(* Visualisation VIS_CHONOEDITOR
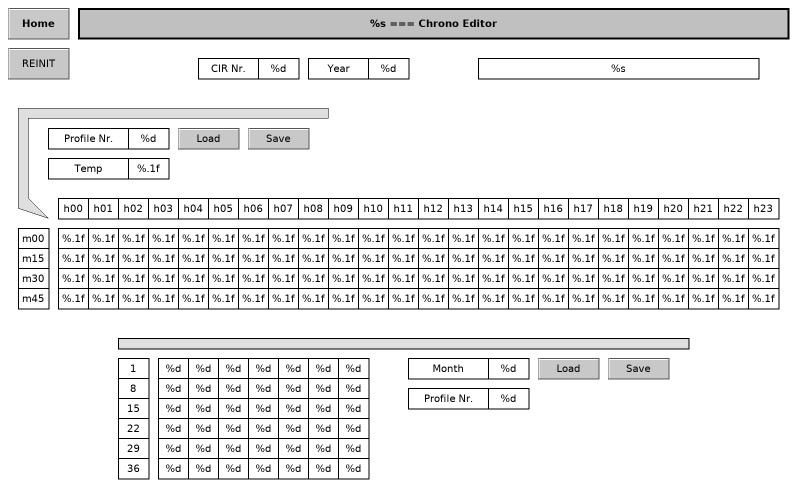
rectangle at (200,60)-(261,81): text "CIR Nr."
rectangle at (260,60)-(301,81): text "%d"; shows CronEd.CN_Sel; alarm colour if CronEd.CN_Sel<>CronEd.CN_Act; editable 1..6
rectangle at (50,130)-(131,151): text "Profile Nr."
rectangle at (130,130)-(171,151): text "%d"; shows CronEd.PR_Sel; alarm colour if CronEd.PR_Sel<>CronEd.PR_Act; editable 1..10
rectangle at (50,160)-(131,181): text "Temp"
rectangle at (130,160)-(171,181): text "%.1f"; shows CronEd.PR_TT; editable
button at (180,130)-(241,151): text "Load"; toggles CronEd.PR_Load
button at (250,130)-(311,151): text "Save"; toggles CronEd.PR_Save
rectangle at (20,230)-(51,251): text "m00"
rectangle at (20,250)-(51,271): text "m15"
rectangle at (20,270)-(51,291): text "m30"
rectangle at (20,290)-(51,311): text "m45"
rectangle at (80,10)-(791,41): text "%s === Chrono Editor"; shows .Plant_NAME
button at (10,10)-(71,41): text "Home"; opens PLC_VISU
rounded rectangle at (60,230)-(91,251): text "%.1f"; shows WORD_TO_REAL(CronEd.PR.Setpoint[0])/10; runs INTERN ASSIGN CronEd.PR.Setpoint[0]:=(REAL_TO_WORD(CronEd.PR_TT*10))
rounded rectangle at (60,250)-(91,271): text "%.1f"; shows WORD_TO_REAL(CronEd.PR.Setpoint[1])/10; runs INTERN ASSIGN CronEd.PR.Setpoint[1]:=(REAL_TO_WORD(CronEd.PR_TT*10))
rounded rectangle at (60,270)-(91,291): text "%.1f"; shows WORD_TO_REAL(CronEd.PR.Setpoint[2])/10; runs INTERN ASSIGN CronEd.PR.Setpoint[2]:=(REAL_TO_WORD(CronEd.PR_TT*10))
rounded rectangle at (60,290)-(91,311): text "%.1f"; shows WORD_TO_REAL(CronEd.PR.Setpoint[3])/10; runs INTERN ASSIGN CronEd.PR.Setpoint[3]:=(REAL_TO_WORD(CronEd.PR_TT*10))
rectangle at (60,200)-(91,221): text "h00"; runs INTERN ASSIGN CronEd.PR.Setpoint[0]:=(REAL_TO_WORD(CronEd.PR_TT*10));INTERN ASSIGN CronEd.PR.Setpoint[1]:=(REAL_TO_WORD(CronEd.PR_TT*10));INTERN ASSIGN CronEd.PR.Setpoint[2]:=(REAL_TO_WORD(CronEd.PR_TT*10));INTERN ASSIGN CronEd.PR.Setpoint[3]:=(REAL_TO_WORD(CronEd.PR_TT*10))
rounded rectangle at (90,230)-(121,251): text "%.1f"; shows WORD_TO_REAL(CronEd.PR.Setpoint[4])/10; runs INTERN ASSIGN CronEd.PR.Setpoint[4]:=(REAL_TO_WORD(CronEd.PR_TT*10))
rounded rectangle at (90,250)-(121,271): text "%.1f"; shows WORD_TO_REAL(CronEd.PR.Setpoint[5])/10; runs INTERN ASSIGN CronEd.PR.Setpoint[5]:=(REAL_TO_WORD(CronEd.PR_TT*10))
rounded rectangle at (90,270)-(121,291): text "%.1f"; shows WORD_TO_REAL(CronEd.PR.Setpoint[6])/10; runs INTERN ASSIGN CronEd.PR.Setpoint[6]:=(REAL_TO_WORD(CronEd.PR_TT*10))
rounded rectangle at (90,290)-(121,311): text "%.1f"; shows WORD_TO_REAL(CronEd.PR.Setpoint[7])/10; runs INTERN ASSIGN CronEd.PR.Setpoint[7]:=(REAL_TO_WORD(CronEd.PR_TT*10))
rectangle at (90,200)-(121,221): text "h01"; runs INTERN ASSIGN CronEd.PR.Setpoint[4]:=(REAL_TO_WORD(CronEd.PR_TT*10));INTERN ASSIGN CronEd.PR.Setpoint[5]:=(REAL_TO_WORD(CronEd.PR_TT*10));INTERN ASSIGN CronEd.PR.Setpoint[6]:=(REAL_TO_WORD(CronEd.PR_TT*10));INTERN ASSIGN CronEd.PR.Setpoint[7]:=(REAL_TO_WORD(CronEd.PR_TT*10))
rounded rectangle at (120,230)-(151,251): text "%.1f"; shows WORD_TO_REAL(CronEd.PR.Setpoint[8])/10; runs INTERN ASSIGN CronEd.PR.Setpoint[8]:=(REAL_TO_WORD(CronEd.PR_TT*10))
rounded rectangle at (120,250)-(151,271): text "%.1f"; shows WORD_TO_REAL(CronEd.PR.Setpoint[9])/10; runs INTERN ASSIGN CronEd.PR.Setpoint[9]:=(REAL_TO_WORD(CronEd.PR_TT*10))
rounded rectangle at (120,270)-(151,291): text "%.1f"; shows WORD_TO_REAL(CronEd.PR.Setpoint[10])/10; runs INTERN ASSIGN CronEd.PR.Setpoint[10]:=(REAL_TO_WORD(CronEd.PR_TT*10))
rounded rectangle at (120,290)-(151,311): text "%.1f"; shows WORD_TO_REAL(CronEd.PR.Setpoint[11])/10; runs INTERN ASSIGN CronEd.PR.Setpoint[11]:=(REAL_TO_WORD(CronEd.PR_TT*10))
rectangle at (120,200)-(151,221): text "h02"; runs INTERN ASSIGN CronEd.PR.Setpoint[8]:=(REAL_TO_WORD(CronEd.PR_TT*10));INTERN ASSIGN CronEd.PR.Setpoint[9]:=(REAL_TO_WORD(CronEd.PR_TT*10));INTERN ASSIGN CronEd.PR.Setpoint[10]:=(REAL_TO_WORD(CronEd.PR_TT*10));INTERN ASSIGN CronEd.PR.Setpoint[11]:=(REAL_TO_WORD(CronEd.PR_TT*10))
rounded rectangle at (150,230)-(181,251): text "%.1f"; shows WORD_TO_REAL(CronEd.PR.Setpoint[12])/10; runs INTERN ASSIGN CronEd.PR.Setpoint[12]:=(REAL_TO_WORD(CronEd.PR_TT*10))
rounded rectangle at (150,250)-(181,271): text "%.1f"; shows WORD_TO_REAL(CronEd.PR.Setpoint[13])/10; runs INTERN ASSIGN CronEd.PR.Setpoint[13]:=(REAL_TO_WORD(CronEd.PR_TT*10))
rounded rectangle at (150,270)-(181,291): text "%.1f"; shows WORD_TO_REAL(CronEd.PR.Setpoint[14])/10; runs INTERN ASSIGN CronEd.PR.Setpoint[14]:=(REAL_TO_WORD(CronEd.PR_TT*10))
rounded rectangle at (150,290)-(181,311): text "%.1f"; shows WORD_TO_REAL(CronEd.PR.Setpoint[15])/10; runs INTERN ASSIGN CronEd.PR.Setpoint[15]:=(REAL_TO_WORD(CronEd.PR_TT*10))
rectangle at (150,200)-(181,221): text "h03"; runs INTERN ASSIGN CronEd.PR.Setpoint[15]:=(REAL_TO_WORD(CronEd.PR_TT*10));INTERN ASSIGN CronEd.PR.Setpoint[14]:=(REAL_TO_WORD(CronEd.PR_TT*10));INTERN ASSIGN CronEd.PR.Setpoint[13]:=(REAL_TO_WORD(CronEd.PR_TT*10));INTERN ASSIGN CronEd.PR.Setpoint[12]:=(REAL_TO_WORD(CronEd.PR_TT*10))
rounded rectangle at (180,230)-(211,251): text "%.1f"; shows WORD_TO_REAL(CronEd.PR.Setpoint[16])/10; runs INTERN ASSIGN CronEd.PR.Setpoint[16]:=(REAL_TO_WORD(CronEd.PR_TT*10))
rounded rectangle at (180,250)-(211,271): text "%.1f"; shows WORD_TO_REAL(CronEd.PR.Setpoint[17])/10; runs INTERN ASSIGN CronEd.PR.Setpoint[17]:=(REAL_TO_WORD(CronEd.PR_TT*10))
rounded rectangle at (180,270)-(211,291): text "%.1f"; shows WORD_TO_REAL(CronEd.PR.Setpoint[18])/10; runs INTERN ASSIGN CronEd.PR.Setpoint[18]:=(REAL_TO_WORD(CronEd.PR_TT*10))
rounded rectangle at (180,290)-(211,311): text "%.1f"; shows WORD_TO_REAL(CronEd.PR.Setpoint[19])/10; runs INTERN ASSIGN CronEd.PR.Setpoint[19]:=(REAL_TO_WORD(CronEd.PR_TT*10))
rectangle at (180,200)-(211,221): text "h04"; runs INTERN ASSIGN CronEd.PR.Setpoint[19]:=(REAL_TO_WORD(CronEd.PR_TT*10));INTERN ASSIGN CronEd.PR.Setpoint[18]:=(REAL_TO_WORD(CronEd.PR_TT*10));INTERN ASSIGN CronEd.PR.Setpoint[17]:=(REAL_TO_WORD(CronEd.PR_TT*10));INTERN ASSIGN CronEd.PR.Setpoint[16]:=(REAL_TO_WORD(CronEd.PR_TT*10))
rounded rectangle at (210,230)-(241,251): text "%.1f"; shows WORD_TO_REAL(CronEd.PR.Setpoint[20])/10; runs INTERN ASSIGN CronEd.PR.Setpoint[20]:=(REAL_TO_WORD(CronEd.PR_TT*10))
rounded rectangle at (210,250)-(241,271): text "%.1f"; shows WORD_TO_REAL(CronEd.PR.Setpoint[21])/10; runs INTERN ASSIGN CronEd.PR.Setpoint[21]:=(REAL_TO_WORD(CronEd.PR_TT*10))
rounded rectangle at (210,270)-(241,291): text "%.1f"; shows WORD_TO_REAL(CronEd.PR.Setpoint[22])/10; runs INTERN ASSIGN CronEd.PR.Setpoint[22]:=(REAL_TO_WORD(CronEd.PR_TT*10))
rounded rectangle at (210,290)-(241,311): text "%.1f"; shows WORD_TO_REAL(CronEd.PR.Setpoint[23])/10; runs INTERN ASSIGN CronEd.PR.Setpoint[23]:=(REAL_TO_WORD(CronEd.PR_TT*10))
rectangle at (210,200)-(241,221): text "h05"; runs INTERN ASSIGN CronEd.PR.Setpoint[23]:=(REAL_TO_WORD(CronEd.PR_TT*10));INTERN ASSIGN CronEd.PR.Setpoint[22]:=(REAL_TO_WORD(CronEd.PR_TT*10));INTERN ASSIGN CronEd.PR.Setpoint[21]:=(REAL_TO_WORD(CronEd.PR_TT*10));INTERN ASSIGN CronEd.PR.Setpoint[20]:=(REAL_TO_WORD(CronEd.PR_TT*10))
rounded rectangle at (240,230)-(271,251): text "%.1f"; shows WORD_TO_REAL(CronEd.PR.Setpoint[24])/10; runs INTERN ASSIGN CronEd.PR.Setpoint[24]:=(REAL_TO_WORD(CronEd.PR_TT*10))
rounded rectangle at (240,250)-(271,271): text "%.1f"; shows WORD_TO_REAL(CronEd.PR.Setpoint[25])/10; runs INTERN ASSIGN CronEd.PR.Setpoint[25]:=(REAL_TO_WORD(CronEd.PR_TT*10))
rounded rectangle at (240,270)-(271,291): text "%.1f"; shows WORD_TO_REAL(CronEd.PR.Setpoint[26])/10; runs INTERN ASSIGN CronEd.PR.Setpoint[26]:=(REAL_TO_WORD(CronEd.PR_TT*10))
rounded rectangle at (240,290)-(271,311): text "%.1f"; shows WORD_TO_REAL(CronEd.PR.Setpoint[27])/10; runs INTERN ASSIGN CronEd.PR.Setpoint[27]:=(REAL_TO_WORD(CronEd.PR_TT*10))
rectangle at (240,200)-(271,221): text "h06"; runs INTERN ASSIGN CronEd.PR.Setpoint[27]:=(REAL_TO_WORD(CronEd.PR_TT*10));INTERN ASSIGN CronEd.PR.Setpoint[26]:=(REAL_TO_WORD(CronEd.PR_TT*10));INTERN ASSIGN CronEd.PR.Setpoint[25]:=(REAL_TO_WORD(CronEd.PR_TT*10));INTERN ASSIGN CronEd.PR.Setpoint[24]:=(REAL_TO_WORD(CronEd.PR_TT*10))
rounded rectangle at (270,230)-(301,251): text "%.1f"; shows WORD_TO_REAL(CronEd.PR.Setpoint[28])/10; runs INTERN ASSIGN CronEd.PR.Setpoint[28]:=(REAL_TO_WORD(CronEd.PR_TT*10))
rounded rectangle at (270,250)-(301,271): text "%.1f"; shows WORD_TO_REAL(CronEd.PR.Setpoint[29])/10; runs INTERN ASSIGN CronEd.PR.Setpoint[29]:=(REAL_TO_WORD(CronEd.PR_TT*10))
rounded rectangle at (270,270)-(301,291): text "%.1f"; shows WORD_TO_REAL(CronEd.PR.Setpoint[30])/10; runs INTERN ASSIGN CronEd.PR.Setpoint[30]:=(REAL_TO_WORD(CronEd.PR_TT*10))
rounded rectangle at (270,290)-(301,311): text "%.1f"; shows WORD_TO_REAL(CronEd.PR.Setpoint[31])/10; runs INTERN ASSIGN CronEd.PR.Setpoint[31]:=(REAL_TO_WORD(CronEd.PR_TT*10))
rectangle at (270,200)-(301,221): text "h07"; runs INTERN ASSIGN CronEd.PR.Setpoint[31]:=(REAL_TO_WORD(CronEd.PR_TT*10));INTERN ASSIGN CronEd.PR.Setpoint[30]:=(REAL_TO_WORD(CronEd.PR_TT*10));INTERN ASSIGN CronEd.PR.Setpoint[29]:=(REAL_TO_WORD(CronEd.PR_TT*10));INTERN ASSIGN CronEd.PR.Setpoint[28]:=(REAL_TO_WORD(CronEd.PR_TT*10))
rounded rectangle at (300,230)-(331,251): text "%.1f"; shows WORD_TO_REAL(CronEd.PR.Setpoint[32])/10; runs INTERN ASSIGN CronEd.PR.Setpoint[32]:=(REAL_TO_WORD(CronEd.PR_TT*10))
rounded rectangle at (300,250)-(331,271): text "%.1f"; shows WORD_TO_REAL(CronEd.PR.Setpoint[33])/10; runs INTERN ASSIGN CronEd.PR.Setpoint[33]:=(REAL_TO_WORD(CronEd.PR_TT*10))
rounded rectangle at (300,270)-(331,291): text "%.1f"; shows WORD_TO_REAL(CronEd.PR.Setpoint[34])/10; runs INTERN ASSIGN CronEd.PR.Setpoint[34]:=(REAL_TO_WORD(CronEd.PR_TT*10))
rounded rectangle at (300,290)-(331,311): text "%.1f"; shows WORD_TO_REAL(CronEd.PR.Setpoint[35])/10; runs INTERN ASSIGN CronEd.PR.Setpoint[35]:=(REAL_TO_WORD(CronEd.PR_TT*10))
rectangle at (300,200)-(331,221): text "h08"; runs INTERN ASSIGN CronEd.PR.Setpoint[35]:=(REAL_TO_WORD(CronEd.PR_TT*10));INTERN ASSIGN CronEd.PR.Setpoint[34]:=(REAL_TO_WORD(CronEd.PR_TT*10));INTERN ASSIGN CronEd.PR.Setpoint[33]:=(REAL_TO_WORD(CronEd.PR_TT*10));INTERN ASSIGN CronEd.PR.Setpoint[32]:=(REAL_TO_WORD(CronEd.PR_TT*10))
rounded rectangle at (330,230)-(361,251): text "%.1f"; shows WORD_TO_REAL(CronEd.PR.Setpoint[36])/10; runs INTERN ASSIGN CronEd.PR.Setpoint[36]:=(REAL_TO_WORD(CronEd.PR_TT*10))
rounded rectangle at (330,250)-(361,271): text "%.1f"; shows WORD_TO_REAL(CronEd.PR.Setpoint[37])/10; runs INTERN ASSIGN CronEd.PR.Setpoint[37]:=(REAL_TO_WORD(CronEd.PR_TT*10))
rounded rectangle at (330,270)-(361,291): text "%.1f"; shows WORD_TO_REAL(CronEd.PR.Setpoint[38])/10; runs INTERN ASSIGN CronEd.PR.Setpoint[38]:=(REAL_TO_WORD(CronEd.PR_TT*10))
rounded rectangle at (330,290)-(361,311): text "%.1f"; shows WORD_TO_REAL(CronEd.PR.Setpoint[39])/10; runs INTERN ASSIGN CronEd.PR.Setpoint[39]:=(REAL_TO_WORD(CronEd.PR_TT*10))
rectangle at (330,200)-(361,221): text "h09"; runs INTERN ASSIGN CronEd.PR.Setpoint[39]:=(REAL_TO_WORD(CronEd.PR_TT*10));INTERN ASSIGN CronEd.PR.Setpoint[38]:=(REAL_TO_WORD(CronEd.PR_TT*10));INTERN ASSIGN CronEd.PR.Setpoint[37]:=(REAL_TO_WORD(CronEd.PR_TT*10));INTERN ASSIGN CronEd.PR.Setpoint[36]:=(REAL_TO_WORD(CronEd.PR_TT*10))
rounded rectangle at (360,230)-(391,251): text "%.1f"; shows WORD_TO_REAL(CronEd.PR.Setpoint[40])/10; runs INTERN ASSIGN CronEd.PR.Setpoint[40]:=(REAL_TO_WORD(CronEd.PR_TT*10))
rounded rectangle at (360,250)-(391,271): text "%.1f"; shows WORD_TO_REAL(CronEd.PR.Setpoint[41])/10; runs INTERN ASSIGN CronEd.PR.Setpoint[41]:=(REAL_TO_WORD(CronEd.PR_TT*10))
rounded rectangle at (360,270)-(391,291): text "%.1f"; shows WORD_TO_REAL(CronEd.PR.Setpoint[42])/10; runs INTERN ASSIGN CronEd.PR.Setpoint[42]:=(REAL_TO_WORD(CronEd.PR_TT*10))
rounded rectangle at (360,290)-(391,311): text "%.1f"; shows WORD_TO_REAL(CronEd.PR.Setpoint[43])/10; runs INTERN ASSIGN CronEd.PR.Setpoint[43]:=(REAL_TO_WORD(CronEd.PR_TT*10))
rectangle at (360,200)-(391,221): text "h10"; runs INTERN ASSIGN CronEd.PR.Setpoint[43]:=(REAL_TO_WORD(CronEd.PR_TT*10));INTERN ASSIGN CronEd.PR.Setpoint[42]:=(REAL_TO_WORD(CronEd.PR_TT*10));INTERN ASSIGN CronEd.PR.Setpoint[41]:=(REAL_TO_WORD(CronEd.PR_TT*10));INTERN ASSIGN CronEd.PR.Setpoint[40]:=(REAL_TO_WORD(CronEd.PR_TT*10))
rounded rectangle at (390,230)-(421,251): text "%.1f"; shows WORD_TO_REAL(CronEd.PR.Setpoint[44])/10; runs INTERN ASSIGN CronEd.PR.Setpoint[44]:=(REAL_TO_WORD(CronEd.PR_TT*10))
rounded rectangle at (390,250)-(421,271): text "%.1f"; shows WORD_TO_REAL(CronEd.PR.Setpoint[45])/10; runs INTERN ASSIGN CronEd.PR.Setpoint[45]:=(REAL_TO_WORD(CronEd.PR_TT*10))
rounded rectangle at (390,270)-(421,291): text "%.1f"; shows WORD_TO_REAL(CronEd.PR.Setpoint[46])/10; runs INTERN ASSIGN CronEd.PR.Setpoint[46]:=(REAL_TO_WORD(CronEd.PR_TT*10))
rounded rectangle at (390,290)-(421,311): text "%.1f"; shows WORD_TO_REAL(CronEd.PR.Setpoint[47])/10; runs INTERN ASSIGN CronEd.PR.Setpoint[47]:=(REAL_TO_WORD(CronEd.PR_TT*10))
rectangle at (390,200)-(421,221): text "h11"; runs INTERN ASSIGN CronEd.PR.Setpoint[47]:=(REAL_TO_WORD(CronEd.PR_TT*10));INTERN ASSIGN CronEd.PR.Setpoint[46]:=(REAL_TO_WORD(CronEd.PR_TT*10));INTERN ASSIGN CronEd.PR.Setpoint[45]:=(REAL_TO_WORD(CronEd.PR_TT*10));INTERN ASSIGN CronEd.PR.Setpoint[44]:=(REAL_TO_WORD(CronEd.PR_TT*10))
rounded rectangle at (420,230)-(451,251): text "%.1f"; shows WORD_TO_REAL(CronEd.PR.Setpoint[48])/10; runs INTERN ASSIGN CronEd.PR.Setpoint[48]:=(REAL_TO_WORD(CronEd.PR_TT*10))
rounded rectangle at (420,250)-(451,271): text "%.1f"; shows WORD_TO_REAL(CronEd.PR.Setpoint[49])/10; runs INTERN ASSIGN CronEd.PR.Setpoint[49]:=(REAL_TO_WORD(CronEd.PR_TT*10))
rounded rectangle at (420,270)-(451,291): text "%.1f"; shows WORD_TO_REAL(CronEd.PR.Setpoint[50])/10; runs INTERN ASSIGN CronEd.PR.Setpoint[50]:=(REAL_TO_WORD(CronEd.PR_TT*10))
rounded rectangle at (420,290)-(451,311): text "%.1f"; shows WORD_TO_REAL(CronEd.PR.Setpoint[51])/10; runs INTERN ASSIGN CronEd.PR.Setpoint[51]:=(REAL_TO_WORD(CronEd.PR_TT*10))
rectangle at (420,200)-(451,221): text "h12"; runs INTERN ASSIGN CronEd.PR.Setpoint[51]:=(REAL_TO_WORD(CronEd.PR_TT*10));INTERN ASSIGN CronEd.PR.Setpoint[50]:=(REAL_TO_WORD(CronEd.PR_TT*10));INTERN ASSIGN CronEd.PR.Setpoint[49]:=(REAL_TO_WORD(CronEd.PR_TT*10));INTERN ASSIGN CronEd.PR.Setpoint[48]:=(REAL_TO_WORD(CronEd.PR_TT*10))
rounded rectangle at (450,230)-(481,251): text "%.1f"; shows WORD_TO_REAL(CronEd.PR.Setpoint[52])/10; runs INTERN ASSIGN CronEd.PR.Setpoint[52]:=(REAL_TO_WORD(CronEd.PR_TT*10))
rounded rectangle at (450,250)-(481,271): text "%.1f"; shows WORD_TO_REAL(CronEd.PR.Setpoint[53])/10; runs INTERN ASSIGN CronEd.PR.Setpoint[53]:=(REAL_TO_WORD(CronEd.PR_TT*10))
rounded rectangle at (450,270)-(481,291): text "%.1f"; shows WORD_TO_REAL(CronEd.PR.Setpoint[54])/10; runs INTERN ASSIGN CronEd.PR.Setpoint[54]:=(REAL_TO_WORD(CronEd.PR_TT*10))
rounded rectangle at (450,290)-(481,311): text "%.1f"; shows WORD_TO_REAL(CronEd.PR.Setpoint[55])/10; runs INTERN ASSIGN CronEd.PR.Setpoint[55]:=(REAL_TO_WORD(CronEd.PR_TT*10))
rectangle at (450,200)-(481,221): text "h13"; runs INTERN ASSIGN CronEd.PR.Setpoint[55]:=(REAL_TO_WORD(CronEd.PR_TT*10));INTERN ASSIGN CronEd.PR.Setpoint[54]:=(REAL_TO_WORD(CronEd.PR_TT*10));INTERN ASSIGN CronEd.PR.Setpoint[53]:=(REAL_TO_WORD(CronEd.PR_TT*10));INTERN ASSIGN CronEd.PR.Setpoint[52]:=(REAL_TO_WORD(CronEd.PR_TT*10))
rounded rectangle at (480,230)-(511,251): text "%.1f"; shows WORD_TO_REAL(CronEd.PR.Setpoint[56])/10; runs INTERN ASSIGN CronEd.PR.Setpoint[56]:=(REAL_TO_WORD(CronEd.PR_TT*10))
rounded rectangle at (480,250)-(511,271): text "%.1f"; shows WORD_TO_REAL(CronEd.PR.Setpoint[57])/10; runs INTERN ASSIGN CronEd.PR.Setpoint[57]:=(REAL_TO_WORD(CronEd.PR_TT*10))
rounded rectangle at (480,270)-(511,291): text "%.1f"; shows WORD_TO_REAL(CronEd.PR.Setpoint[58])/10; runs INTERN ASSIGN CronEd.PR.Setpoint[58]:=(REAL_TO_WORD(CronEd.PR_TT*10))
rounded rectangle at (480,290)-(511,311): text "%.1f"; shows WORD_TO_REAL(CronEd.PR.Setpoint[59])/10; runs INTERN ASSIGN CronEd.PR.Setpoint[59]:=(REAL_TO_WORD(CronEd.PR_TT*10))
rectangle at (480,200)-(511,221): text "h14"; runs INTERN ASSIGN CronEd.PR.Setpoint[59]:=(REAL_TO_WORD(CronEd.PR_TT*10));INTERN ASSIGN CronEd.PR.Setpoint[58]:=(REAL_TO_WORD(CronEd.PR_TT*10));INTERN ASSIGN CronEd.PR.Setpoint[57]:=(REAL_TO_WORD(CronEd.PR_TT*10));INTERN ASSIGN CronEd.PR.Setpoint[56]:=(REAL_TO_WORD(CronEd.PR_TT*10))
rounded rectangle at (510,230)-(541,251): text "%.1f"; shows WORD_TO_REAL(CronEd.PR.Setpoint[60])/10; runs INTERN ASSIGN CronEd.PR.Setpoint[60]:=(REAL_TO_WORD(CronEd.PR_TT*10))
rounded rectangle at (510,250)-(541,271): text "%.1f"; shows WORD_TO_REAL(CronEd.PR.Setpoint[61])/10; runs INTERN ASSIGN CronEd.PR.Setpoint[61]:=(REAL_TO_WORD(CronEd.PR_TT*10))
rounded rectangle at (510,270)-(541,291): text "%.1f"; shows WORD_TO_REAL(CronEd.PR.Setpoint[62])/10; runs INTERN ASSIGN CronEd.PR.Setpoint[62]:=(REAL_TO_WORD(CronEd.PR_TT*10))
rounded rectangle at (510,290)-(541,311): text "%.1f"; shows WORD_TO_REAL(CronEd.PR.Setpoint[63])/10; runs INTERN ASSIGN CronEd.PR.Setpoint[63]:=(REAL_TO_WORD(CronEd.PR_TT*10))
rectangle at (510,200)-(541,221): text "h15"; runs INTERN ASSIGN CronEd.PR.Setpoint[63]:=(REAL_TO_WORD(CronEd.PR_TT*10));INTERN ASSIGN CronEd.PR.Setpoint[62]:=(REAL_TO_WORD(CronEd.PR_TT*10));INTERN ASSIGN CronEd.PR.Setpoint[61]:=(REAL_TO_WORD(CronEd.PR_TT*10));INTERN ASSIGN CronEd.PR.Setpoint[60]:=(REAL_TO_WORD(CronEd.PR_TT*10))
rounded rectangle at (540,230)-(571,251): text "%.1f"; shows WORD_TO_REAL(CronEd.PR.Setpoint[64])/10; runs INTERN ASSIGN CronEd.PR.Setpoint[64]:=(REAL_TO_WORD(CronEd.PR_TT*10))
rounded rectangle at (540,250)-(571,271): text "%.1f"; shows WORD_TO_REAL(CronEd.PR.Setpoint[65])/10; runs INTERN ASSIGN CronEd.PR.Setpoint[65]:=(REAL_TO_WORD(CronEd.PR_TT*10))
rounded rectangle at (540,270)-(571,291): text "%.1f"; shows WORD_TO_REAL(CronEd.PR.Setpoint[66])/10; runs INTERN ASSIGN CronEd.PR.Setpoint[66]:=(REAL_TO_WORD(CronEd.PR_TT*10))
rounded rectangle at (540,290)-(571,311): text "%.1f"; shows WORD_TO_REAL(CronEd.PR.Setpoint[67])/10; runs INTERN ASSIGN CronEd.PR.Setpoint[67]:=(REAL_TO_WORD(CronEd.PR_TT*10))
rectangle at (540,200)-(571,221): text "h16"; runs INTERN ASSIGN CronEd.PR.Setpoint[67]:=(REAL_TO_WORD(CronEd.PR_TT*10));INTERN ASSIGN CronEd.PR.Setpoint[66]:=(REAL_TO_WORD(CronEd.PR_TT*10));INTERN ASSIGN CronEd.PR.Setpoint[65]:=(REAL_TO_WORD(CronEd.PR_TT*10));INTERN ASSIGN CronEd.PR.Setpoint[64]:=(REAL_TO_WORD(CronEd.PR_TT*10))
rounded rectangle at (570,230)-(601,251): text "%.1f"; shows WORD_TO_REAL(CronEd.PR.Setpoint[68])/10; runs INTERN ASSIGN CronEd.PR.Setpoint[68]:=(REAL_TO_WORD(CronEd.PR_TT*10))
rounded rectangle at (570,250)-(601,271): text "%.1f"; shows WORD_TO_REAL(CronEd.PR.Setpoint[69])/10; runs INTERN ASSIGN CronEd.PR.Setpoint[69]:=(REAL_TO_WORD(CronEd.PR_TT*10))
rounded rectangle at (570,270)-(601,291): text "%.1f"; shows WORD_TO_REAL(CronEd.PR.Setpoint[70])/10; runs INTERN ASSIGN CronEd.PR.Setpoint[70]:=(REAL_TO_WORD(CronEd.PR_TT*10))
rounded rectangle at (570,290)-(601,311): text "%.1f"; shows WORD_TO_REAL(CronEd.PR.Setpoint[71])/10; runs INTERN ASSIGN CronEd.PR.Setpoint[71]:=(REAL_TO_WORD(CronEd.PR_TT*10))
rectangle at (570,200)-(601,221): text "h17"; runs INTERN ASSIGN CronEd.PR.Setpoint[71]:=(REAL_TO_WORD(CronEd.PR_TT*10));INTERN ASSIGN CronEd.PR.Setpoint[70]:=(REAL_TO_WORD(CronEd.PR_TT*10));INTERN ASSIGN CronEd.PR.Setpoint[69]:=(REAL_TO_WORD(CronEd.PR_TT*10));INTERN ASSIGN CronEd.PR.Setpoint[68]:=(REAL_TO_WORD(CronEd.PR_TT*10))
rounded rectangle at (600,230)-(631,251): text "%.1f"; shows WORD_TO_REAL(CronEd.PR.Setpoint[72])/10; runs INTERN ASSIGN CronEd.PR.Setpoint[72]:=(REAL_TO_WORD(CronEd.PR_TT*10))
rounded rectangle at (600,250)-(631,271): text "%.1f"; shows WORD_TO_REAL(CronEd.PR.Setpoint[73])/10; runs INTERN ASSIGN CronEd.PR.Setpoint[73]:=(REAL_TO_WORD(CronEd.PR_TT*10))
rounded rectangle at (600,270)-(631,291): text "%.1f"; shows WORD_TO_REAL(CronEd.PR.Setpoint[74])/10; runs INTERN ASSIGN CronEd.PR.Setpoint[74]:=(REAL_TO_WORD(CronEd.PR_TT*10))
rounded rectangle at (600,290)-(631,311): text "%.1f"; shows WORD_TO_REAL(CronEd.PR.Setpoint[75])/10; runs INTERN ASSIGN CronEd.PR.Setpoint[75]:=(REAL_TO_WORD(CronEd.PR_TT*10))
rectangle at (600,200)-(631,221): text "h18"; runs INTERN ASSIGN CronEd.PR.Setpoint[75]:=(REAL_TO_WORD(CronEd.PR_TT*10));INTERN ASSIGN CronEd.PR.Setpoint[74]:=(REAL_TO_WORD(CronEd.PR_TT*10));INTERN ASSIGN CronEd.PR.Setpoint[73]:=(REAL_TO_WORD(CronEd.PR_TT*10));INTERN ASSIGN CronEd.PR.Setpoint[72]:=(REAL_TO_WORD(CronEd.PR_TT*10))
rounded rectangle at (630,230)-(661,251): text "%.1f"; shows WORD_TO_REAL(CronEd.PR.Setpoint[76])/10; runs INTERN ASSIGN CronEd.PR.Setpoint[76]:=(REAL_TO_WORD(CronEd.PR_TT*10))
rounded rectangle at (630,250)-(661,271): text "%.1f"; shows WORD_TO_REAL(CronEd.PR.Setpoint[77])/10; runs INTERN ASSIGN CronEd.PR.Setpoint[77]:=(REAL_TO_WORD(CronEd.PR_TT*10))
rounded rectangle at (630,270)-(661,291): text "%.1f"; shows WORD_TO_REAL(CronEd.PR.Setpoint[78])/10; runs INTERN ASSIGN CronEd.PR.Setpoint[78]:=(REAL_TO_WORD(CronEd.PR_TT*10))
rounded rectangle at (630,290)-(661,311): text "%.1f"; shows WORD_TO_REAL(CronEd.PR.Setpoint[79])/10; runs INTERN ASSIGN CronEd.PR.Setpoint[79]:=(REAL_TO_WORD(CronEd.PR_TT*10))
rectangle at (630,200)-(661,221): text "h19"; runs INTERN ASSIGN CronEd.PR.Setpoint[79]:=(REAL_TO_WORD(CronEd.PR_TT*10));INTERN ASSIGN CronEd.PR.Setpoint[78]:=(REAL_TO_WORD(CronEd.PR_TT*10));INTERN ASSIGN CronEd.PR.Setpoint[77]:=(REAL_TO_WORD(CronEd.PR_TT*10));INTERN ASSIGN CronEd.PR.Setpoint[76]:=(REAL_TO_WORD(CronEd.PR_TT*10))
rounded rectangle at (660,230)-(691,251): text "%.1f"; shows WORD_TO_REAL(CronEd.PR.Setpoint[80])/10; runs INTERN ASSIGN CronEd.PR.Setpoint[80]:=(REAL_TO_WORD(CronEd.PR_TT*10))
rounded rectangle at (660,250)-(691,271): text "%.1f"; shows WORD_TO_REAL(CronEd.PR.Setpoint[81])/10; runs INTERN ASSIGN CronEd.PR.Setpoint[81]:=(REAL_TO_WORD(CronEd.PR_TT*10))
rounded rectangle at (660,270)-(691,291): text "%.1f"; shows WORD_TO_REAL(CronEd.PR.Setpoint[82])/10; runs INTERN ASSIGN CronEd.PR.Setpoint[82]:=(REAL_TO_WORD(CronEd.PR_TT*10))
rounded rectangle at (660,290)-(691,311): text "%.1f"; shows WORD_TO_REAL(CronEd.PR.Setpoint[83])/10; runs INTERN ASSIGN CronEd.PR.Setpoint[83]:=(REAL_TO_WORD(CronEd.PR_TT*10))
rectangle at (660,200)-(691,221): text "h20"; runs INTERN ASSIGN CronEd.PR.Setpoint[83]:=(REAL_TO_WORD(CronEd.PR_TT*10));INTERN ASSIGN CronEd.PR.Setpoint[82]:=(REAL_TO_WORD(CronEd.PR_TT*10));INTERN ASSIGN CronEd.PR.Setpoint[81]:=(REAL_TO_WORD(CronEd.PR_TT*10));INTERN ASSIGN CronEd.PR.Setpoint[80]:=(REAL_TO_WORD(CronEd.PR_TT*10))
rounded rectangle at (690,230)-(721,251): text "%.1f"; shows WORD_TO_REAL(CronEd.PR.Setpoint[84])/10; runs INTERN ASSIGN CronEd.PR.Setpoint[84]:=(REAL_TO_WORD(CronEd.PR_TT*10))
rounded rectangle at (690,250)-(721,271): text "%.1f"; shows WORD_TO_REAL(CronEd.PR.Setpoint[85])/10; runs INTERN ASSIGN CronEd.PR.Setpoint[85]:=(REAL_TO_WORD(CronEd.PR_TT*10))
rounded rectangle at (690,270)-(721,291): text "%.1f"; shows WORD_TO_REAL(CronEd.PR.Setpoint[86])/10; runs INTERN ASSIGN CronEd.PR.Setpoint[86]:=(REAL_TO_WORD(CronEd.PR_TT*10))
rounded rectangle at (690,290)-(721,311): text "%.1f"; shows WORD_TO_REAL(CronEd.PR.Setpoint[87])/10; runs INTERN ASSIGN CronEd.PR.Setpoint[87]:=(REAL_TO_WORD(CronEd.PR_TT*10))
rectangle at (690,200)-(721,221): text "h21"; runs INTERN ASSIGN CronEd.PR.Setpoint[87]:=(REAL_TO_WORD(CronEd.PR_TT*10));INTERN ASSIGN CronEd.PR.Setpoint[86]:=(REAL_TO_WORD(CronEd.PR_TT*10));INTERN ASSIGN CronEd.PR.Setpoint[85]:=(REAL_TO_WORD(CronEd.PR_TT*10));INTERN ASSIGN CronEd.PR.Setpoint[84]:=(REAL_TO_WORD(CronEd.PR_TT*10))
rounded rectangle at (720,230)-(751,251): text "%.1f"; shows WORD_TO_REAL(CronEd.PR.Setpoint[88])/10; runs INTERN ASSIGN CronEd.PR.Setpoint[88]:=(REAL_TO_WORD(CronEd.PR_TT*10))
rounded rectangle at (720,250)-(751,271): text "%.1f"; shows WORD_TO_REAL(CronEd.PR.Setpoint[89])/10; runs INTERN ASSIGN CronEd.PR.Setpoint[89]:=(REAL_TO_WORD(CronEd.PR_TT*10))
rounded rectangle at (720,270)-(751,291): text "%.1f"; shows WORD_TO_REAL(CronEd.PR.Setpoint[90])/10; runs INTERN ASSIGN CronEd.PR.Setpoint[90]:=(REAL_TO_WORD(CronEd.PR_TT*10))
rounded rectangle at (720,290)-(751,311): text "%.1f"; shows WORD_TO_REAL(CronEd.PR.Setpoint[91])/10; runs INTERN ASSIGN CronEd.PR.Setpoint[91]:=(REAL_TO_WORD(CronEd.PR_TT*10))
rectangle at (720,200)-(751,221): text "h22"; runs INTERN ASSIGN CronEd.PR.Setpoint[91]:=(REAL_TO_WORD(CronEd.PR_TT*10));INTERN ASSIGN CronEd.PR.Setpoint[90]:=(REAL_TO_WORD(CronEd.PR_TT*10));INTERN ASSIGN CronEd.PR.Setpoint[89]:=(REAL_TO_WORD(CronEd.PR_TT*10));INTERN ASSIGN CronEd.PR.Setpoint[88]:=(REAL_TO_WORD(CronEd.PR_TT*10))
rounded rectangle at (750,230)-(781,251): text "%.1f"; shows WORD_TO_REAL(CronEd.PR.Setpoint[92])/10; runs INTERN ASSIGN CronEd.PR.Setpoint[92]:=(REAL_TO_WORD(CronEd.PR_TT*10))
rounded rectangle at (750,250)-(781,271): text "%.1f"; shows WORD_TO_REAL(CronEd.PR.Setpoint[93])/10; runs INTERN ASSIGN CronEd.PR.Setpoint[93]:=(REAL_TO_WORD(CronEd.PR_TT*10))
rounded rectangle at (750,270)-(781,291): text "%.1f"; shows WORD_TO_REAL(CronEd.PR.Setpoint[94])/10; runs INTERN ASSIGN CronEd.PR.Setpoint[94]:=(REAL_TO_WORD(CronEd.PR_TT*10))
rounded rectangle at (750,290)-(781,311): text "%.1f"; shows WORD_TO_REAL(CronEd.PR.Setpoint[95])/10; runs INTERN ASSIGN CronEd.PR.Setpoint[95]:=(REAL_TO_WORD(CronEd.PR_TT*10))
rectangle at (750,200)-(781,221): text "h23"; runs INTERN ASSIGN CronEd.PR.Setpoint[95]:=(REAL_TO_WORD(CronEd.PR_TT*10));INTERN ASSIGN CronEd.PR.Setpoint[94]:=(REAL_TO_WORD(CronEd.PR_TT*10));INTERN ASSIGN CronEd.PR.Setpoint[93]:=(REAL_TO_WORD(CronEd.PR_TT*10));INTERN ASSIGN CronEd.PR.Setpoint[92]:=(REAL_TO_WORD(CronEd.PR_TT*10))
rectangle at (410,360)-(491,381): text "Month"
rectangle at (490,360)-(531,381): text "%d"; shows CronEd.CA_Sel; alarm colour if CronEd.CA_Sel<>CronEd.CA_Act; editable 1..12
rectangle at (410,390)-(491,411): text "Profile Nr."
rectangle at (490,390)-(531,411): text "%d"; shows CronEd.CA_TPR; editable 0..10
button at (540,360)-(601,381): text "Load"; toggles CronEd.CA_Load
button at (610,360)-(671,381): text "Save"; toggles CronEd.CA_Save
rounded rectangle at (160,360)-(191,381): text "%d"; shows CronEd.CA.Profile[0]; invisible if CronEd.CA_DayF>0; alarm colour if CronEd.CA.Profile[0]=0; runs INTERN ASSIGN CronEd.CA.Profile[0]:=(CronEd.CA_TPR)
rectangle at (120,360)-(151,381): text "1"
rounded rectangle at (190,360)-(221,381): text "%d"; shows CronEd.CA.Profile[1]; invisible if CronEd.CA_DayF>1; alarm colour if CronEd.CA.Profile[1]=0; runs INTERN ASSIGN CronEd.CA.Profile[1]:=(CronEd.CA_TPR)
rounded rectangle at (220,360)-(251,381): text "%d"; shows CronEd.CA.Profile[2]; invisible if CronEd.CA_DayF>2; alarm colour if CronEd.CA.Profile[2]=0; runs INTERN ASSIGN CronEd.CA.Profile[2]:=(CronEd.CA_TPR)
rounded rectangle at (250,360)-(281,381): text "%d"; shows CronEd.CA.Profile[3]; invisible if CronEd.CA_DayF>3; alarm colour if CronEd.CA.Profile[3]=0; runs INTERN ASSIGN CronEd.CA.Profile[3]:=(CronEd.CA_TPR)
rounded rectangle at (280,360)-(311,381): text "%d"; shows CronEd.CA.Profile[4]; invisible if CronEd.CA_DayF>4; alarm colour if CronEd.CA.Profile[4]=0; runs INTERN ASSIGN CronEd.CA.Profile[4]:=(CronEd.CA_TPR)
rounded rectangle at (310,360)-(341,381): text "%d"; shows CronEd.CA.Profile[5]; invisible if CronEd.CA_DayF>5; alarm colour if CronEd.CA.Profile[5]=0; runs INTERN ASSIGN CronEd.CA.Profile[5]:=(CronEd.CA_TPR)
rounded rectangle at (340,360)-(371,381): text "%d"; shows CronEd.CA.Profile[6]; alarm colour if CronEd.CA.Profile[6]=0; runs INTERN ASSIGN CronEd.CA.Profile[6]:=(CronEd.CA_TPR)
rounded rectangle at (160,380)-(191,401): text "%d"; shows CronEd.CA.Profile[7]; alarm colour if CronEd.CA.Profile[7]=0; runs INTERN ASSIGN CronEd.CA.Profile[7]:=(CronEd.CA_TPR)
rectangle at (120,380)-(151,401): text "8"
rounded rectangle at (190,380)-(221,401): text "%d"; shows CronEd.CA.Profile[8]; alarm colour if CronEd.CA.Profile[8]=0; runs INTERN ASSIGN CronEd.CA.Profile[8]:=(CronEd.CA_TPR)
rounded rectangle at (220,380)-(251,401): text "%d"; shows CronEd.CA.Profile[9]; alarm colour if CronEd.CA.Profile[9]=0; runs INTERN ASSIGN CronEd.CA.Profile[9]:=(CronEd.CA_TPR)
rounded rectangle at (250,380)-(281,401): text "%d"; shows CronEd.CA.Profile[10]; alarm colour if CronEd.CA.Profile[10]=0; runs INTERN ASSIGN CronEd.CA.Profile[10]:=(CronEd.CA_TPR)
rounded rectangle at (280,380)-(311,401): text "%d"; shows CronEd.CA.Profile[11]; alarm colour if CronEd.CA.Profile[11]=0; runs INTERN ASSIGN CronEd.CA.Profile[11]:=(CronEd.CA_TPR)
rounded rectangle at (310,380)-(341,401): text "%d"; shows CronEd.CA.Profile[12]; alarm colour if CronEd.CA.Profile[12]=0; runs INTERN ASSIGN CronEd.CA.Profile[12]:=(CronEd.CA_TPR)
rounded rectangle at (340,380)-(371,401): text "%d"; shows CronEd.CA.Profile[13]; alarm colour if CronEd.CA.Profile[13]=0; runs INTERN ASSIGN CronEd.CA.Profile[13]:=(CronEd.CA_TPR)
rounded rectangle at (160,400)-(191,421): text "%d"; shows CronEd.CA.Profile[14]; alarm colour if CronEd.CA.Profile[14]=0; runs INTERN ASSIGN CronEd.CA.Profile[14]:=(CronEd.CA_TPR)
rectangle at (120,400)-(151,421): text "15"
rounded rectangle at (190,400)-(221,421): text "%d"; shows CronEd.CA.Profile[15]; alarm colour if CronEd.CA.Profile[15]=0; runs INTERN ASSIGN CronEd.CA.Profile[15]:=(CronEd.CA_TPR)
rounded rectangle at (220,400)-(251,421): text "%d"; shows CronEd.CA.Profile[16]; alarm colour if CronEd.CA.Profile[16]=0; runs INTERN ASSIGN CronEd.CA.Profile[16]:=(CronEd.CA_TPR)
rounded rectangle at (250,400)-(281,421): text "%d"; shows CronEd.CA.Profile[17]; alarm colour if CronEd.CA.Profile[17]=0; runs INTERN ASSIGN CronEd.CA.Profile[17]:=(CronEd.CA_TPR)
rounded rectangle at (280,400)-(311,421): text "%d"; shows CronEd.CA.Profile[18]; alarm colour if CronEd.CA.Profile[18]=0; runs INTERN ASSIGN CronEd.CA.Profile[18]:=(CronEd.CA_TPR)
rounded rectangle at (310,400)-(341,421): text "%d"; shows CronEd.CA.Profile[19]; alarm colour if CronEd.CA.Profile[19]=0; runs INTERN ASSIGN CronEd.CA.Profile[19]:=(CronEd.CA_TPR)
rounded rectangle at (340,400)-(371,421): text "%d"; shows CronEd.CA.Profile[20]; alarm colour if CronEd.CA.Profile[20]=0; runs INTERN ASSIGN CronEd.CA.Profile[20]:=(CronEd.CA_TPR)
rounded rectangle at (160,420)-(191,441): text "%d"; shows CronEd.CA.Profile[21]; alarm colour if CronEd.CA.Profile[21]=0; runs INTERN ASSIGN CronEd.CA.Profile[21]:=(CronEd.CA_TPR)
rectangle at (120,420)-(151,441): text "22"
rounded rectangle at (190,420)-(221,441): text "%d"; shows CronEd.CA.Profile[22]; alarm colour if CronEd.CA.Profile[22]=0; runs INTERN ASSIGN CronEd.CA.Profile[22]:=(CronEd.CA_TPR)
rounded rectangle at (220,420)-(251,441): text "%d"; shows CronEd.CA.Profile[23]; alarm colour if CronEd.CA.Profile[23]=0; runs INTERN ASSIGN CronEd.CA.Profile[23]:=(CronEd.CA_TPR)
rounded rectangle at (250,420)-(281,441): text "%d"; shows CronEd.CA.Profile[24]; alarm colour if CronEd.CA.Profile[24]=0; runs INTERN ASSIGN CronEd.CA.Profile[24]:=(CronEd.CA_TPR)
rounded rectangle at (280,420)-(311,441): text "%d"; shows CronEd.CA.Profile[25]; alarm colour if CronEd.CA.Profile[25]=0; runs INTERN ASSIGN CronEd.CA.Profile[25]:=(CronEd.CA_TPR)
rounded rectangle at (310,420)-(341,441): text "%d"; shows CronEd.CA.Profile[26]; alarm colour if CronEd.CA.Profile[26]=0; runs INTERN ASSIGN CronEd.CA.Profile[26]:=(CronEd.CA_TPR)
rounded rectangle at (340,420)-(371,441): text "%d"; shows CronEd.CA.Profile[27]; alarm colour if CronEd.CA.Profile[27]=0; runs INTERN ASSIGN CronEd.CA.Profile[27]:=(CronEd.CA_TPR)
rounded rectangle at (160,440)-(191,461): text "%d"; shows CronEd.CA.Profile[28]; alarm colour if CronEd.CA.Profile[28]=0; runs INTERN ASSIGN CronEd.CA.Profile[28]:=(CronEd.CA_TPR)
rectangle at (120,440)-(151,461): text "29"
rounded rectangle at (190,440)-(221,461): text "%d"; shows CronEd.CA.Profile[29]; alarm colour if CronEd.CA.Profile[29]=0; runs INTERN ASSIGN CronEd.CA.Profile[29]:=(CronEd.CA_TPR)
rounded rectangle at (220,440)-(251,461): text "%d"; shows CronEd.CA.Profile[30]; alarm colour if CronEd.CA.Profile[30]=0; runs INTERN ASSIGN CronEd.CA.Profile[30]:=(CronEd.CA_TPR)
rounded rectangle at (250,440)-(281,461): text "%d"; shows CronEd.CA.Profile[31]; alarm colour if CronEd.CA.Profile[31]=0; runs INTERN ASSIGN CronEd.CA.Profile[31]:=(CronEd.CA_TPR)
rounded rectangle at (280,440)-(311,461): text "%d"; shows CronEd.CA.Profile[32]; invisible if CronEd.CA_DayL<32; alarm colour if CronEd.CA.Profile[32]=0; runs INTERN ASSIGN CronEd.CA.Profile[32]:=(CronEd.CA_TPR)
rounded rectangle at (310,440)-(341,461): text "%d"; shows CronEd.CA.Profile[33]; invisible if CronEd.CA_DayL<33; alarm colour if CronEd.CA.Profile[33]=0; runs INTERN ASSIGN CronEd.CA.Profile[33]:=(CronEd.CA_TPR)
rounded rectangle at (340,440)-(371,461): text "%d"; shows CronEd.CA.Profile[34]; invisible if CronEd.CA_DayL<34; alarm colour if CronEd.CA.Profile[34]=0; runs INTERN ASSIGN CronEd.CA.Profile[34]:=(CronEd.CA_TPR)
rounded rectangle at (160,460)-(191,481): text "%d"; shows CronEd.CA.Profile[35]; invisible if CronEd.CA_DayL<35; alarm colour if CronEd.CA.Profile[35]=0; runs INTERN ASSIGN CronEd.CA.Profile[35]:=(CronEd.CA_TPR)
rectangle at (120,460)-(151,481): text "36"; invisible if CronEd.CA_DayL<35
rounded rectangle at (190,460)-(221,481): text "%d"; shows CronEd.CA.Profile[36]; invisible if CronEd.CA_DayL<36; alarm colour if CronEd.CA.Profile[36]=0; runs INTERN ASSIGN CronEd.CA.Profile[36]:=(CronEd.CA_TPR)
rounded rectangle at (220,460)-(251,481): text "%d"; shows CronEd.CA.Profile[37]; invisible if CronEd.CA_DayL<37; alarm colour if CronEd.CA.Profile[37]=0; runs INTERN ASSIGN CronEd.CA.Profile[37]:=(CronEd.CA_TPR)
rounded rectangle at (250,460)-(281,481): text "%d"; shows CronEd.CA.Profile[38]; invisible if CronEd.CA_DayL<38; alarm colour if CronEd.CA.Profile[38]=0; runs INTERN ASSIGN CronEd.CA.Profile[38]:=(CronEd.CA_TPR)
rounded rectangle at (280,460)-(311,481): text "%d"; shows CronEd.CA.Profile[39]; invisible if CronEd.CA_DayL<39; alarm colour if CronEd.CA.Profile[39]=0; runs INTERN ASSIGN CronEd.CA.Profile[39]:=(CronEd.CA_TPR)
rounded rectangle at (310,460)-(341,481): text "%d"; shows CronEd.CA.Profile[40]; invisible if CronEd.CA_DayL<40; alarm colour if CronEd.CA.Profile[40]=0; runs INTERN ASSIGN CronEd.CA.Profile[40]:=(CronEd.CA_TPR)
rounded rectangle at (340,460)-(371,481): text "%d"; shows CronEd.CA.Profile[41]; invisible if CronEd.CA_DayL<41; alarm colour if CronEd.CA.Profile[41]=0; runs INTERN ASSIGN CronEd.CA.Profile[41]:=(CronEd.CA_TPR)
rectangle at (310,60)-(371,81): text "Year"
rectangle at (370,60)-(411,81): text "%d"; shows CronEd.CN_YSel; alarm colour if CronEd.CN_YSel<>CronEd.CN_YAct; editable 2000..2100
rectangle at (480,60)-(761,81): text "%s"; shows CronEd.Message
button at (10,50)-(71,81): text "REINIT"; runs INTERN ASSIGN THER01.InitOK:=(FALSE);INTERN ASSIGN THER02.InitOK:=(FALSE);INTERN ASSIGN THER03.InitOK:=(FALSE);INTERN ASSIGN THER04.InitOK:=(FALSE)
2 more shapes without text or variables
*)

(* Visualisation VIS_VRD01
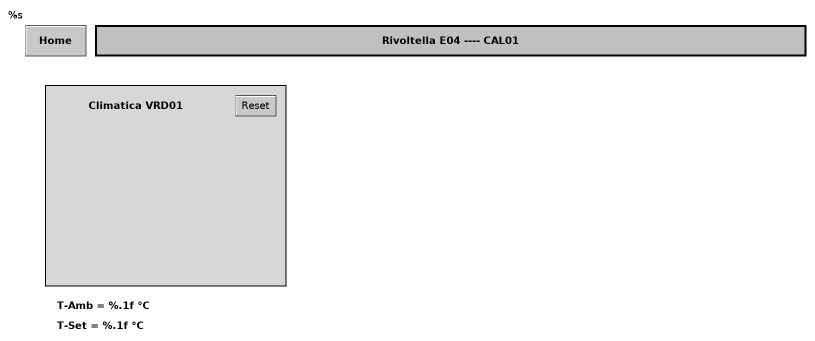
rectangle at (0,0)-(0,0): text "%s"; shows VRD01_Clima.Points[INDEX].X; invisible if INDEX>4; editable
rectangle at (0,0)-(0,0): text "%s"; shows VRD01_Clima.Points[INDEX].Y; invisible if INDEX>4; editable
rectangle at (40,80)-(201,101): text "Climatica VRD01"
button at (220,80)-(261,101): text "Reset"; runs INTERN ASSIGN VRD01_Clima.InitOK:=(FALSE)
button at (10,10)-(71,41): text "Home"; opens PLC_VISU
rectangle at (40,300)-(181,321): text "T-Set = %.1f °C"; shows INT_TO_REAL(.VRD01.Ctrl_SetPoint)/10
rectangle at (40,280)-(181,301): text "T-Amb = %.1f °C"; shows INT_TO_REAL(.T_AMB)/10; alarm colour if T_AMB>2000
rectangle at (80,10)-(791,41): text "Rivoltella E04 ---- CAL01"
1 more shapes without text or variables
*)

(* Visualisation VIS_VRD02
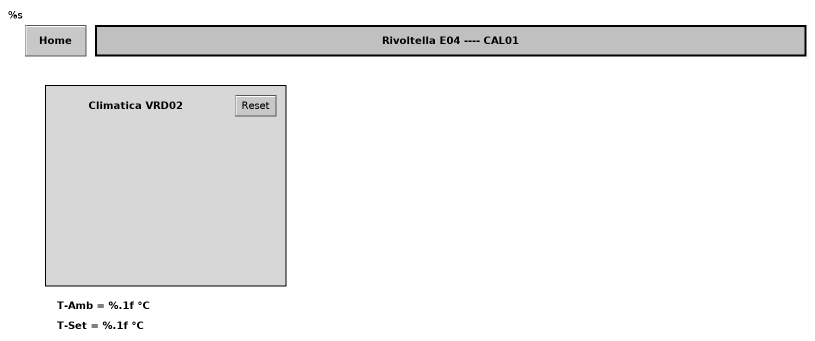
rectangle at (0,0)-(0,0): text "%s"; shows VRD02_Clima.Points[INDEX].X; invisible if INDEX>4; editable
rectangle at (0,0)-(0,0): text "%s"; shows VRD02_Clima.Points[INDEX].Y; invisible if INDEX>4; editable
rectangle at (40,80)-(201,101): text "Climatica VRD02"
button at (220,80)-(261,101): text "Reset"; runs INTERN ASSIGN VRD02_Clima.InitOK:=(FALSE)
button at (10,10)-(71,41): text "Home"; opens PLC_VISU
rectangle at (40,300)-(181,321): text "T-Set = %.1f °C"; shows INT_TO_REAL(.VRD02.Ctrl_SetPoint)/10
rectangle at (40,280)-(181,301): text "T-Amb = %.1f °C"; shows INT_TO_REAL(.T_AMB)/10; alarm colour if T_AMB>2000
rectangle at (80,10)-(791,41): text "Rivoltella E04 ---- CAL01"
1 more shapes without text or variables
*)
